TYPE Uc_EventLogTable :
STRUCT
	astEvents			: ARRAY[0..nMaxEvents] OF ST_EventOutput;

	bQuitt				: BOOL;
	nIdx				: INT;	
	
	bAckn				: BOOL;
	bMute				: BOOL;
END_STRUCT
END_TYPE

(* stored: Version 1.1.0.1
   DUT Uc_EventLogTable: Id {4a173722-3366-4944-b612-c29006197e34} *)
